// LS Electric XG5000 project: ㅠ접점을 쓰는이유
// PLC NewPLC
// module base 0 slot 0: 입출력 모듈:XBC-DR20S (DC 24V 입력 12점, 릴레이 출력 8점)

PROGRAM NewProgram (task: 스캔 프로그램)

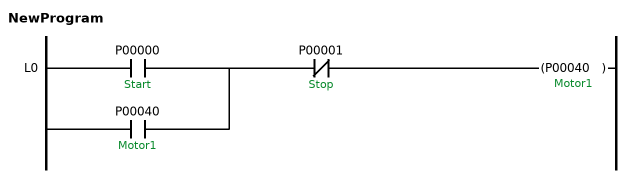
; L0
LOAD      P00000	// Start
OR        P00040	// Motor1
AND NOT   P00001	// Stop
OUT       P00040	// Motor1